FUNCTION_BLOCK FB_ConveyorEntry_ST
VAR_INPUT
END_VAR
VAR_OUTPUT
END_VAR
VAR
	step : INT;
	RtrigInitTrigger : R_TRIG;
	initTrigger : BOOL := TRUE;
	
	eMitterTimer : Tc2_Standard.TP;
	startEmitting : BOOL;
	
END_VAR
VAR_IN_OUT
	control_data : PlantAndCMs.Udt_PlantControl_Mode_1;
	
	control_data_vision : CM_Vision_UDT;
	control_data_Conveyor1 : CM_DO_UDT;
	
	control_data_StopBlade : CM_DO_UDT;
	control_data_emitter : CM_DO_UDT;
END_VAR

RtrigInitTrigger(CLK :=initTrigger);

eMitterTimer(IN := StartEmitting, pt := T#0.2S);


CASE step OF 
	0 : // Init
	
		IF control_data.Auto_Out THEN
			initTrigger := FALSE;
			step := 1;
		END_IF
	
	1: // Step 1 start machine
		
		IF control_data.Startet_Out THEN
			initTrigger := TRUE;
			step := 2;
		END_IF
	2:			
		
		IF control_data_vision.PO_PV = 0 THEN
			startEmitting := TRUE;
			step := 5;
		END_IF
	
	5: 
		startEmitting := FALSE;
		GVL.readyForSorting := FALSE;
		GVL.SortingDone := FALSE;
		
		IF control_data_vision.PO_PV = 1 THEN
			GVL.BLUE_TOP := TRUE;
			GVL.BLUE_BOTTOM := FALSE;
			GVL.BLUE_MIDDLE := FALSE;
			GVL.GREEN_TOP := FALSE;
			GVL.GREEN_BOTTOM := FALSE;
			GVL.GREEN_MIDDLE := FALSE;
			step := 11;
		END_IF
		IF control_data_vision.PO_PV = 2 THEN
			GVL.BLUE_TOP := FALSE;
			GVL.BLUE_BOTTOM := TRUE;
			GVL.BLUE_MIDDLE := FALSE;
			GVL.GREEN_TOP := FALSE;
			GVL.GREEN_BOTTOM := FALSE;
			GVL.GREEN_MIDDLE := FALSE;
			step := 11;
		END_IF
		IF control_data_vision.PO_PV = 3 THEN
			GVL.BLUE_TOP := FALSE;
			GVL.BLUE_BOTTOM := FALSE;
			GVL.BLUE_MIDDLE := TRUE;
			GVL.GREEN_TOP := FALSE;
			GVL.GREEN_BOTTOM := FALSE;
			GVL.GREEN_MIDDLE := FALSE;
			step := 11;
		END_IF
		IF control_data_vision.PO_PV = 4 THEN
			GVL.BLUE_TOP := FALSE;
			GVL.BLUE_BOTTOM := FALSE;
			GVL.BLUE_MIDDLE := FALSE;
			GVL.GREEN_TOP := TRUE;
			GVL.GREEN_BOTTOM := FALSE;
			GVL.GREEN_MIDDLE := FALSE;
			step := 11;
		END_IF
		IF control_data_vision.PO_PV = 5 THEN
			GVL.BLUE_TOP := FALSE;
			GVL.BLUE_BOTTOM := FALSE;
			GVL.BLUE_MIDDLE := FALSE;
			GVL.GREEN_TOP := FALSE;
			GVL.GREEN_BOTTOM := TRUE;
			GVL.GREEN_MIDDLE := FALSE;
			step := 11;
		END_IF
		IF control_data_vision.PO_PV = 6 THEN
			GVL.BLUE_TOP := FALSE;
			GVL.BLUE_BOTTOM := FALSE;
			GVL.BLUE_MIDDLE := FALSE;
			GVL.GREEN_TOP := FALSE;
			GVL.GREEN_BOTTOM := FALSE;
			GVL.GREEN_MIDDLE := TRUE;
			step := 11;
		END_IF
		

	11:
		GVL.readyForSorting := TRUE;
		
		IF GVL.SortingDone THEN
			GVL.BLUE_TOP := FALSE;
			GVL.BLUE_BOTTOM := FALSE;
			GVL.BLUE_MIDDLE := FALSE;
			GVL.GREEN_TOP := FALSE;
			GVL.GREEN_BOTTOM := FALSE;
			GVL.GREEN_MIDDLE := FALSE;
			
			startEmitting := TRUE;
			
			step := 2;
		END_IF
		
END_CASE


control_data_emitter.PO_HighCommand := eMitterTimer.Q;

control_data_Conveyor1.PO_HighCommand := control_data.Startet_Out;

END_FUNCTION_BLOCK

(* stored: Version 1.1.0.1, ProductVersion 3.1.4024.13
   POU FB_ConveyorEntry_ST: Id {f2d86c63-254e-4119-8c51-2f80b74ae540}, SpecialFunc None *)
